// TIA Portal project "TIA-Portal-ModbusTCPExample" (V16)

(* hardware
DEVICE "S7-1200-Station_1"  S7-1200 Station
   slot 0: "Baugruppenträger_0"  S7-1200 Rack  Rack  V1.0
   slot 1: "PLC_1"  CPU 1211C DC/DC/DC  6ES7 211-1AE40-0XB0  V4.1
*)

// ===== PLC "PLC_1"  CPU 1211C DC/DC/DC =====

DATA_BLOCK "Modbus_TCON"   // DB2
{ S7_Optimized_Access := 'TRUE' }
VERSION : 0.1
   VAR
      TCON : TCON_IP_v4;
   END_VAR
BEGIN
   TCON.ID := 1;
   TCON.LocalPort := 502;
   TCON.InterfaceId := 64;
END_DATA_BLOCK

DATA_BLOCK "HoldingReg"   // DB3
{ S7_Optimized_Access := 'TRUE' }
VERSION : 0.1
   VAR
      MB_Reg1 : Int;
      MB_Reg2 : Int;
      MB_reg3 : Int;
   END_VAR
BEGIN
END_DATA_BLOCK

ORGANIZATION_BLOCK "Main"   // OB1, FBD, ProgramCycle
TITLE = "Main Program Sweep (Cycle)"
{ S7_Optimized_Access := 'TRUE' }
VERSION : 0.1
   VAR_INPUT
      Initial_Call : Bool;   // Initial call of this OB
      Remanence : Bool;   // =True, if remanent data are available
   END_VAR
BEGIN

REGION Network 1
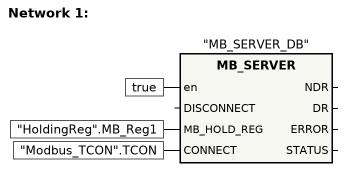
   IF true THEN
       "MB_SERVER_DB"(MB_HOLD_REG := "HoldingReg".MB_Reg1, CONNECT := "Modbus_TCON".TCON);   // MB_SERVER
   END_IF;
END_REGION
END_ORGANIZATION_BLOCK